Fanuc KAREL source: kt00835.compact.KL

PROGRAM KT00835
%STACKSIZE=65535
%PRIORITY=65535
%NOLOCKGROUP
VAR
R1 : REAL
R2 : REAL
OUT : REAL
BEGIN
R1=2.0
R2=3.0
R1=2.0
R2=3.0
OUT=SQRT(R1)
END KT00835
